ABB RAPID module: Module1.mod

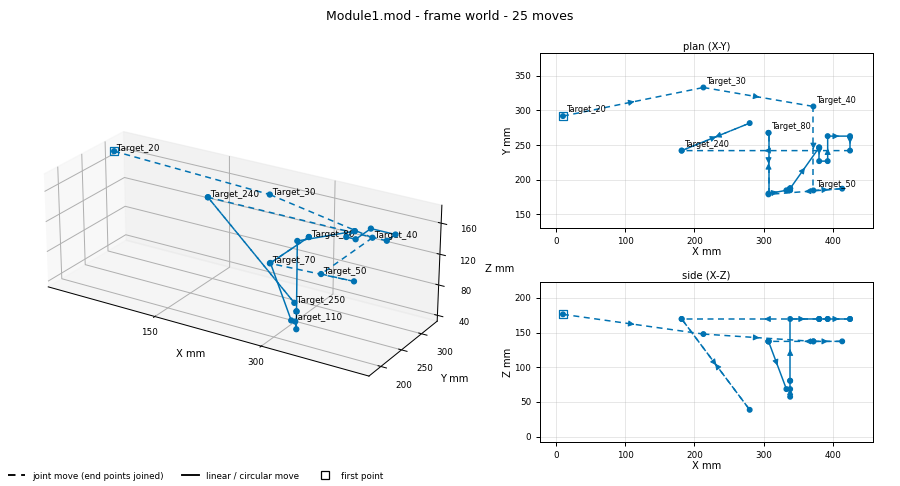
[picture p0: tool path of Module1.mod in frame world, 25 of 25 moves have a stored position in this frame; points joined in program order, loops and branches not executed]
MODULE Module1

	CONST robtarget Target_10:=[[419.170322148,249.802548244,191.497848229],[0.040124088,-0.583044032,0.811344151,0.01305309],[0,1,-1,4],[-122.717189906,9E+09,9E+09,9E+09,9E+09,9E+09]];
	CONST robtarget Target_20:=[[10.457656172,291.807433463,176.354847091],[0.248288991,0.071063339,-0.705346937,0.660142618],[0,-1,0,4],[163.797976426,9E+09,9E+09,9E+09,9E+09,9E+09]];
	CONST robtarget Target_30:=[[212.888290668,333.048761883,147.91359348],[0.066010621,0.842421125,-0.111215182,0.523068283],[0,-1,0,4],[163.797976918,9E+09,9E+09,9E+09,9E+09,9E+09]];
	CONST robtarget Target_40:=[[371.422593942,305.712173822,137.388797672],[0.457279618,-0.51920164,0.460433877,-0.556170525],[-1,-1,1,4],[164.810337123,9E+09,9E+09,9E+09,9E+09,9E+09]];
	CONST robtarget Target_50:=[[371.422669025,184.656495549,137.388730749],[0.45727955,-0.519201612,0.460434087,-0.556170434],[-1,-1,1,4],[164.81033427,9E+09,9E+09,9E+09,9E+09,9E+09]];
	CONST robtarget Target_60:=[[412.939496836,187.197681679,137.388418149],[0.457279325,-0.519201634,0.460434592,-0.55617018],[-1,-1,1,4],[164.810337118,9E+09,9E+09,9E+09,9E+09,9E+09]];
	CONST robtarget Target_70:=[[306.715986743,178.95899168,137.388245956],[0.457279164,-0.519201608,0.460434877,-0.5561701],[-1,-1,1,4],[164.810333683,9E+09,9E+09,9E+09,9E+09,9E+09]];
	CONST robtarget Target_80:=[[306.716114229,267.673696389,137.388188332],[0.457279158,-0.519201531,0.460435085,-0.556170005],[-1,-1,1,4],[164.810336018,9E+09,9E+09,9E+09,9E+09,9E+09]];
	CONST robtarget Target_90:=[[306.716414573,267.674145085,137.38817767],[0.034383048,0.760763487,-0.648014557,-0.011569673],[0,-3,3,4],[164.810336639,9E+09,9E+09,9E+09,9E+09,9E+09]];
	CONST robtarget Target_100:=[[306.71653824,180.120525812,137.388160421],[0.034382982,0.760763498,-0.648014545,-0.011569813],[-1,-3,2,4],[164.810332395,9E+09,9E+09,9E+09,9E+09,9E+09]];
	CONST robtarget Target_110:=[[332.520883703,184.866836739,68.574286274],[0.034382546,0.76076337,-0.648014697,-0.011570999],[-1,-3,2,4],[164.810341689,9E+09,9E+09,9E+09,9E+09,9E+09]];
	CONST robtarget Target_120:=[[337.926742079,184.866994086,68.574258233],[0.034382626,0.760763329,-0.648014738,-0.01157119],[-1,-3,2,4],[164.810332747,9E+09,9E+09,9E+09,9E+09,9E+09]];
	CONST robtarget Target_130:=[[337.92674638,187.492031839,57.550963112],[0.034382637,0.760763244,-0.648014829,-0.011571579],[-1,-3,2,4],[164.810331376,9E+09,9E+09,9E+09,9E+09,9E+09]];
	CONST robtarget Target_140:=[[337.92675862,187.492169056,80.592893178],[0.034382757,0.760763265,-0.648014795,-0.011571748],[-1,-3,2,4],[164.810332212,9E+09,9E+09,9E+09,9E+09,9E+09]];
	CONST robtarget Target_150:=[[337.926758615,187.492169056,80.592893178],[0.018524543,0.999330732,0.0046913,-0.031191676],[-1,-3,1,4],[164.810332212,9E+09,9E+09,9E+09,9E+09,9E+09]];
	CONST robtarget Target_160:=[[337.926790343,187.49236794,169.665764789],[0.01852449,0.999330728,0.004691285,-0.031191852],[-1,-3,1,4],[164.8103333,9E+09,9E+09,9E+09,9E+09,9E+09]];
	CONST robtarget Target_170:=[[379.779612425,246.655988999,169.665450165],[0.018523946,0.999330723,0.004691051,-0.031192362],[-1,-3,2,4],[162.186368156,9E+09,9E+09,9E+09,9E+09,9E+09]];
	CONST robtarget Target_180:=[[379.779612425,246.655988999,169.665450165],[0.018523946,0.999330723,0.004691051,-0.031192362],[-1,-3,2,4],[162.186368156,9E+09,9E+09,9E+09,9E+09,9E+09]];
	CONST robtarget Target_190:=[[379.779691233,226.899765789,169.665441657],[0.018523879,0.999330717,0.004691023,-0.031192589],[-1,-3,2,4],[162.186366766,9E+09,9E+09,9E+09,9E+09,9E+09]];
	CONST robtarget Target_200:=[[391.996281361,226.899957165,169.665339804],[0.018523857,0.999330711,0.004690951,-0.031192807],[-1,-3,2,4],[162.186367083,9E+09,9E+09,9E+09,9E+09,9E+09]];
	CONST robtarget Target_210:=[[391.99642781,262.948698629,169.665260033],[0.018523698,0.999330711,0.004690846,-0.031192923],[-1,-3,2,4],[162.186366738,9E+09,9E+09,9E+09,9E+09,9E+09]];
	CONST robtarget Target_220:=[[424.232645938,262.948871742,169.665252544],[0.01852357,0.999330711,0.004690772,-0.031193008],[-1,-3,2,4],[162.186364964,9E+09,9E+09,9E+09,9E+09,9E+09]];
	CONST robtarget Target_230:=[[424.232733766,242.062877627,169.665144176],[0.018523422,0.99933071,0.004690745,-0.031193136],[-1,-3,2,4],[162.18636532,9E+09,9E+09,9E+09,9E+09,9E+09]];
	CONST robtarget Target_240:=[[181.547716343,242.063108437,169.665105208],[0.018523325,0.999330707,0.004690727,-0.031193299],[0,-2,2,4],[162.186364777,9E+09,9E+09,9E+09,9E+09,9E+09]];
	CONST robtarget Target_250:=[[279.584607709,281.698627222,38.725086521],[0.018523011,0.9993307,0.004690539,-0.031193734],[-1,-3,2,4],[162.186368118,9E+09,9E+09,9E+09,9E+09,9E+09]];
	CONST robtarget Target_240_2:=[[181.547716343,242.063108437,169.665105208],[0.018523325,0.999330707,0.004690727,-0.031193299],[0,-2,2,4],[162.186364777,9E+09,9E+09,9E+09,9E+09,9E+09]];
	PROC main()
	    Path_10;
	ENDPROC
	PROC Path_10()
	    MoveJ Target_20,v1000,z100,Servo_2\WObj:=wobj0;
	    MoveJ Target_30,v1000,z100,Servo_2\WObj:=wobj0;
	    MoveJ Target_40,v1000,z100,Servo_2\WObj:=wobj0;
	    MoveJ Target_50,v1000,z100,Servo_2\WObj:=wobj0;
	    MoveJ Target_60,v1000,z100,Servo_2\WObj:=wobj0;
	    WaitTime 2;
	    MoveJ Target_70,v1000,z100,Servo_2\WObj:=wobj0;
	    MoveJ Target_80,v1000,z100,Servo_2\WObj:=wobj0;
	    MoveL Target_90,v1000,z100,Servo_2\WObj:=wobj0;
	    MoveL Target_100,v80,fine,Servo_2\WObj:=wobj0;
	    MoveL Target_110,v1000,z100,Servo_2\WObj:=wobj0;
	    MoveL Target_120,v1000,z100,Servo_2\WObj:=wobj0;
	    MoveL Target_130,v80,fine,Servo_2\WObj:=wobj0;
	    PulseDO attach_ring2;
	    WaitTime 1;
	    MoveL Target_140,v1000,z100,Servo_2\WObj:=wobj0;
	    MoveL Target_150,v1000,z100,Servo_2\WObj:=wobj0;
	    MoveL Target_160,v1000,z100,Servo_2\WObj:=wobj0;
	    MoveL Target_170,v1000,z100,Servo_2\WObj:=wobj0;
	    MoveL Target_180,v1000,z100,Servo_2\WObj:=wobj0;
	    MoveL Target_190,v1000,z100,Servo_2\WObj:=wobj0;
	    MoveL Target_200,v1000,z100,Servo_2\WObj:=wobj0;
	    MoveL Target_210,v1000,z100,Servo_2\WObj:=wobj0;
	    MoveL Target_220,v1000,z100,Servo_2\WObj:=wobj0;
	    MoveL Target_230,v1000,z100,Servo_2\WObj:=wobj0;
	    MoveJ Target_240,v80,fine,Servo_2\WObj:=wobj0;
		MoveJ Target_250,v80,z100,Servo_2\WObj:=wobj0;
		WaitTime 2;
		PulseDO detach_ring2;
		WaitTime 2;
		MoveJ Target_240_2,v80,fine,Servo_2\WObj:=wobj0;
	ENDPROC
ENDMODULE
